// TIA Portal V20 export
TYPE "UDT_Service_Procedure"
   STRUCT
      ProcedureEnable { ExternalAccessible := 'False'; ExternalVisible := 'False'; ExternalWritable := 'False'; S7_SetPoint := 'True'} : "UDT_Service_ProcedureEnable";
   END_STRUCT;
END_TYPE
